// Library/POUs/Trigger/MC_SetTriggerError/Structures/SetTriggerErrorRecvData
{attribute 'pack_mode' := '1'} 
// ------------------------------------------------------------------------- 
//  SRCI Robot Library                                                
// ------------------------------------------------------------------------- 
//                                                                           
//  Object:      SetTriggerErrorRecvData                                       
//  Author:      Thorsten Brach                                                
//  Date:        2024-08-03
//
//  Description:                                              
//   
//                                                                           
//  Copyright: 
//    (C) 2024 Thorsten Brach. All rights reserved                                                                                                                                            
//             Licensed under the LGPL-3.0 license.
//                                                                           
//  Disclaimer:                                                                           
//    This project is provided without any guarantee and can be used for   
//    private and commercial purposes. Any use is at the user’s 
//    own risk and responsibility.
//
// -------------------------------------------------------------------------
TYPE SetTriggerErrorRecvData EXTENDS RspHeader :
STRUCT
  /// Relates to ListenerID >0
  /// Number of successful trigger-based command invocations - For more information refer TO chapter 5.5.12.4
  InvocationCounter : USINT;  
  /// Reserve
  Reserve           : SINT;
  /// Unique system-generated ID of the "Action" when the function is triggered.
  /// • >0: The "Action" is started by the trigger funcrion with identical FollowID.
  /// • <0: The "Action" is stopped by the trigger function with identical FollowID.
  /// For more information see chapter 5.5.12.4 EmitterID, ListenerID, FollowID and OriginID
  OriginID          : INT;
END_STRUCT
END_TYPE

// Library/POUs/Trigger/MC_SetTriggerError/Structures/SetTriggerErrorSendData
{attribute 'pack_mode' := '1'}
// ------------------------------------------------------------------------- 
//  SRCI Robot Library                                                
// ------------------------------------------------------------------------- 
//                                                                           
//  Object:      SetTriggerErrorSendData                                       
//  Author:      Thorsten Brach                                                
//  Date:        2024-08-03
//
//  Description:                                              
//   
//                                                                           
//  Copyright: 
//    (C) 2024 Thorsten Brach. All rights reserved                                                                                                                                            
//             Licensed under the LGPL-3.0 license.
//                                                                           
//  Disclaimer:                                                                           
//    This project is provided without any guarantee and can be used for   
//    private and commercial purposes. Any use is at the user’s 
//    own risk and responsibility.
//
// -------------------------------------------------------------------------
TYPE SetTriggerErrorSendData EXTENDS CmdHeader: 
STRUCT
  /// ID of Action that will be executed when this command is active
  /// • >0: Start Action - Start executing the Action function with the identical ListenerID.
  /// • <0: Stop Action  -  Stop executing the Action function with the identical ListenerID.
  /// • 0: No trigger (default)-  If no EmitterID is defined, the function will not trigger any Action during its execution
  /// For more information see section Triggers of this chapter or chapter 5.5.12.4.
  EmitterID                  : ARRAY [0..3] OF SINT;  
  /// ID of associated trigger function:
  /// • 0: Immediately (default) - Start executing this function immediately.
  /// • >0: Trigger -  Start executing, when the trigger function with the identical EmitterID is triggered.
  /// Always positive.
  /// For more information, see chapter 5.5.12 Triggers
  ListenerID                 : SINT;
  /// Reserve
  Reserve                    : SINT;
  /// Defines error origin through which the associated Action will be triggered
  Mode                       : SINT;
  /// Defines if parametrization messages are included (relates to Mode 0 to 5)
  /// • FALSE (default): Do not include incorrect parametrization
  /// • TRUE: Include incorrect parametrization
  IncludeParameterValidation : BOOL;
  /// Defines message codes through which the associated Action will be triggered (relates to Mode 6 and 7)
  MessageCodes               : ARRAY [0..RobotLibraryParameter.MESSAGE_CODES_MAX] OF DWORD;  
END_STRUCT
END_TYPE

// Library/POUs/Trigger/MC_SetTriggerLimit/Structures/SetTriggerLimitOutCmd
{attribute 'pack_mode' := '1'} 
// ------------------------------------------------------------------------- 
//  SRCI Robot Library                                                
// ------------------------------------------------------------------------- 
//                                                                           
//  Object:      SetTriggerLimitOutCmd                                       
//  Author:      Thorsten Brach                                                
//  Date:        2024-08-03
//
//  Description:                                              
//   
//                                                                           
//  Copyright: 
//    (C) 2024 Thorsten Brach. All rights reserved                                                                                                                                            
//             Licensed under the LGPL-3.0 license.
//                                                                           
//  Disclaimer:                                                                           
//    This project is provided without any guarantee and can be used for   
//    private and commercial purposes. Any use is at the user’s 
//    own risk and responsibility.
//
// -------------------------------------------------------------------------
TYPE SetTriggerLimitOutCmd :
STRUCT
  /// Unique system-generated ID of the "Action" when the function is triggered.
  /// • >0: The "Action" is started by the trigger function with identical FollowID.
  /// • <0: The "Action" is stopped by the trigger function with identical FollowID.
  /// For more information see chapter 5.5.12.4 EmitterID, ListenerID, FollowID and OriginID
  OriginID               : INT;
  /// Relates to ListenerID >0
  /// Number of successful trigger -based command invocations
  /// For more information refer to chapter 5.5.12.4.
  InvocationCounter      : USINT;
  /// Unique system-generated ID of the trigger function when the function is called by user.
  /// For more information see chapter 5.5.12.4.
  FollowID               : DINT;  
END_STRUCT
END_TYPE

// Library/POUs/Trigger/MC_SetTriggerLimit/Structures/SetTriggerLimitParCmd
{attribute 'pack_mode' := '1'} 
// ------------------------------------------------------------------------- 
//  SRCI Robot Library                                                
// ------------------------------------------------------------------------- 
//                                                                           
//  Object:      SetTriggerLimitParCmd                                       
//  Author:      Thorsten Brach                                                
//  Date:        2024-08-03
//
//  Description:                                              
//   
//                                                                           
//  Copyright: 
//    (C) 2024 Thorsten Brach. All rights reserved                                                                                                                                            
//             Licensed under the LGPL-3.0 license.
//                                                                           
//  Disclaimer:                                                                           
//    This project is provided without any guarantee and can be used for   
//    private and commercial purposes. Any use is at the user’s 
//    own risk and responsibility.
//
// -------------------------------------------------------------------------
TYPE SetTriggerLimitParCmd :
STRUCT
  /// Specifies the trigger event by exceeding of the following limit values (one of the following options must be supported)
  TriggerMode            : TriggerModeLimit;
  /// Determines whether the start condition is evaluated or not.
  /// • FALSE: Start condition is not evaluated (default).
  /// • TRUE: Start condition is evaluated
  EvaluateStartCondition : BOOL;
  /// If the tolerance limits for the respective actual data values from the RC are exceeded, the Action function that will be executed.
  /// For "TriggerMode" 1, 2 and 4 the tolerance limits must be entered as follows:
  /// • [0..5]: relates to axes 1 to 6
  /// • [6..11]: relates to external axes 1 to 6.
  /// For "TriggerMode" 3 the tolerance limits must be entered as follows:
  /// • [0]: Following Error in mm.
  /// • [1..11]: Undefined and not relevant.
  /// For all array entries default: 999999
  Data_1                 : ARRAY[0..11] OF REAL;
  /// If the respective actual data values from the RC are under the defined limit, the Action function will be stopped.
  /// For "TriggerMode" 1, 2 and 4 the tolerance limits must be entered as follows:
  /// • [0..5]: relates to axes 1 to 6.
  /// • [6..11]: relates to external axes 1 to 6.
  /// For "TriggerMode" 3 the tolerance limits must be entered as follows:
  /// • [0]: Following Error in mm.
  /// • [1..11]: Undefined and not relevant.
  /// For all array entries default: 999999
  Data_2                 : ARRAY[0..11] OF REAL;
  /// ID of associated trigger function:
  /// • 0: Immediately (default) - Start executing this function immediately.
  /// • >0: Trigger -  Start executing, when the trigger function with the identical EmitterID is triggered.
  /// Always positive.
  /// For more information, see chapter 5.5.12 Triggers
  ListenerID             : SINT;
  /// ID of the Action function that will be executed when the trigger condition is met
  /// • >0: Start Action        - Start executing the Action function with the identical ListenerID.
  /// • <0: Stop Action         - Stop executing the Action function with the identical ListenerID.
  /// •  0: Undefined (default) - If no EmitterID is defined, the function returns an error message
  /// For more information see chapter 5.5.12.4
  EmitterID              : SINT;   
END_STRUCT
END_TYPE

// Library/POUs/Trigger/MC_SetTriggerLimit/Structures/SetTriggerLimitRecvData
{attribute 'pack_mode' := '1'} 
// ------------------------------------------------------------------------- 
//  SRCI Robot Library                                                
// ------------------------------------------------------------------------- 
//                                                                           
//  Object:      SetTriggerLimitRecvData                                       
//  Author:      Thorsten Brach                                                
//  Date:        2024-08-03
//
//  Description:                                              
//   
//                                                                           
//  Copyright: 
//    (C) 2024 Thorsten Brach. All rights reserved                                                                                                                                            
//             Licensed under the LGPL-3.0 license.
//                                                                           
//  Disclaimer:                                                                           
//    This project is provided without any guarantee and can be used for   
//    private and commercial purposes. Any use is at the user’s 
//    own risk and responsibility.
//
// -------------------------------------------------------------------------
TYPE SetTriggerLimitRecvData EXTENDS RspHeader :
STRUCT
  /// Relates to ListenerID >0
  /// Number of successful trigger -based command invocations
  /// For more information refer to chapter 5.5.12.4.
  InvocationCounter      : USINT;
  /// Reserve
  Reserve                : SINT;
  /// Unique system-generated ID of the "Action" when the function is triggered.
  /// • >0: The "Action" is started by the trigger function with identical FollowID.
  /// • <0: The "Action" is stopped by the trigger function with identical FollowID.
  /// For more information see chapter 5.5.12.4 EmitterID, ListenerID, FollowID and OriginID
  OriginID               : INT;
  /// The respective actual data values from the RC that depend on "TriggerMode".
  Data                   : ARRAY [0..11] OF REAL;  
END_STRUCT
END_TYPE

// Library/POUs/Trigger/MC_SetTriggerLimit/Structures/SetTriggerLimitSendData
{attribute 'pack_mode' := '1'}
// ------------------------------------------------------------------------- 
//  SRCI Robot Library                                                
// ------------------------------------------------------------------------- 
//                                                                           
//  Object:      SetTriggerLimitSendData                                       
//  Author:      Thorsten Brach                                                
//  Date:        2024-08-03
//
//  Description:                                              
//   
//                                                                           
//  Copyright: 
//    (C) 2024 Thorsten Brach. All rights reserved                                                                                                                                            
//             Licensed under the LGPL-3.0 license.
//                                                                           
//  Disclaimer:                                                                           
//    This project is provided without any guarantee and can be used for   
//    private and commercial purposes. Any use is at the user’s 
//    own risk and responsibility.
//
// -------------------------------------------------------------------------
TYPE SetTriggerLimitSendData EXTENDS CmdHeader: 
STRUCT
  /// ID of Action that will be executed when this command is active
  /// • >0: Start Action - Start executing the Action function with the identical ListenerID.
  /// • <0: Stop Action  -  Stop executing the Action function with the identical ListenerID.
  /// • 0: No trigger (default)-  If no EmitterID is defined, the function will not trigger any Action during its execution
  /// For more information see section Triggers of this chapter or chapter 5.5.12.4.
  EmitterID              : ARRAY [0..3] OF SINT;  
  /// ID of associated trigger function:
  /// • 0: Immediately (default) - Start executing this function immediately.
  /// • >0: Trigger -  Start executing, when the trigger function with the identical EmitterID is triggered.
  /// Always positive.
  /// For more information, see chapter 5.5.12 Triggers
  ListenerID             : SINT;
  /// If the tolerance limits for the respective actual data values from the RC are exceeded, the Action function that will be executed.
  /// For "TriggerMode" 1, 2 and 4 the tolerance limits must be entered as follows:
  /// • [0..5]: relates to axes 1 to 6
  /// • [6..11]: relates to external axes 1 to 6.
  /// For "TriggerMode" 3 the tolerance limits must be entered as follows:
  /// • [0]: Following Error in mm.
  /// • [1..11]: Undefined and not relevant.
  /// For all array entries default: 999999
  Data_1                 : ARRAY[0..11] OF REAL;
  /// If the respective actual data values from the RC are under the defined limit, the Action function will be stopped.
  /// For "TriggerMode" 1, 2 and 4 the tolerance limits must be entered as follows:
  /// • [0..5]: relates to axes 1 to 6.
  /// • [6..11]: relates to external axes 1 to 6.
  /// For "TriggerMode" 3 the tolerance limits must be entered as follows:
  /// • [0]: Following Error in mm.
  /// • [1..11]: Undefined and not relevant.
  /// For all array entries default: 999999
  Data_2                 : ARRAY[0..11] OF REAL;
  /// Specifies the trigger event by exceeding of the following limit values (one of the following options must be supported)
  TriggerMode            : SINT;
  /// Determines whether the start condition is evaluated or not.
  /// • FALSE: Start condition is not evaluated (default).
  /// • TRUE: Start condition is evaluated
  EvaluateStartCondition : BOOL;
END_STRUCT
END_TYPE

// Library/POUs/Trigger/MC_SetTriggerMotion/Structures/SetTriggerMotionOutCmd
{attribute 'pack_mode' := '1'} 
// ------------------------------------------------------------------------- 
//  SRCI Robot Library                                                
// ------------------------------------------------------------------------- 
//                                                                           
//  Object:      SetTriggerMotionOutCmd                                       
//  Author:      Thorsten Brach                                                
//  Date:        2024-08-03
//
//  Description:                                              
//   
//                                                                           
//  Copyright: 
//    (C) 2024 Thorsten Brach. All rights reserved                                                                                                                                            
//             Licensed under the LGPL-3.0 license.
//                                                                           
//  Disclaimer:                                                                           
//    This project is provided without any guarantee and can be used for   
//    private and commercial purposes. Any use is at the user’s 
//    own risk and responsibility.
//
// -------------------------------------------------------------------------
TYPE SetTriggerMotionOutCmd :
STRUCT
  /// Unique system-generated ID of the "Action" when the function is triggered.
  /// • >0: The "Action" is started by the trigger function with identical FollowID.
  /// • <0: The "Action" is stopped by the trigger function with identical FollowID.
  /// For more information see chapter 5.5.12.4 EmitterID, ListenerID, FollowID and OriginID
  OriginID               : INT;
  /// Relates to ListenerID >0
  /// Number of successful trigger -based command invocations
  /// For more information refer to chapter 5.5.12.4.
  InvocationCounter      : USINT;
  /// Unique system-generated ID of the trigger function when the function is called by user.
  /// For more information see chapter 5.5.12.4.
  FollowID               : DINT;
END_STRUCT
END_TYPE

// Library/POUs/Trigger/MC_SetTriggerMotion/Structures/SetTriggerMotionParCmd
{attribute 'pack_mode' := '1'} 
// ------------------------------------------------------------------------- 
//  SRCI Robot Library                                                
// ------------------------------------------------------------------------- 
//                                                                           
//  Object:      SetTriggerMotionParCmd                                       
//  Author:      Thorsten Brach                                                
//  Date:        2024-08-03
//
//  Description:                                              
//   
//                                                                           
//  Copyright: 
//    (C) 2024 Thorsten Brach. All rights reserved                                                                                                                                            
//             Licensed under the LGPL-3.0 license.
//                                                                           
//  Disclaimer:                                                                           
//    This project is provided without any guarantee and can be used for   
//    private and commercial purposes. Any use is at the user’s 
//    own risk and responsibility.
//
// -------------------------------------------------------------------------
TYPE SetTriggerMotionParCmd :
STRUCT
  ///Defines the trigger condition on which the related Action function will be started:
  TriggerMode_1          : TriggerCondition;
  /// This parameter depends on the input parameter "TriggerMode_1":
  /// • 1: Distance value of trajectory in %.
  /// • 2: Distance value of trajectory in mm.
  /// • 3: TCP velocity value of reference velocity in %
  /// • 4: TCP velocity value of reference velocity in mm.
  /// • 5: Time in ms
  /// The value of the parameter must be positive  
  TriggerParameter_1     : REAL;
  ///Defines the trigger condition on which the related Action function will be started:
  TriggerMode_2          : TriggerCondition;
  /// This parameter depends on the input parameter "TriggerMode_1":
  /// • 1: Distance value of trajectory in %. 
  /// • 2: Distance value of trajectory in mm.
  /// • 3: TCP velocity value of reference velocity in %
  /// • 4: TCP velocity value of reference velocity in mm.
  /// • 5: Time in ms
  /// The value of the parameter must be positive  
  TriggerParameter_2     : REAL;
  /// ID of associated trigger function:
  /// • 0: Immediately (default) - Start executing this function immediately.
  /// • >0: Trigger -  Start executing, when the trigger function with the identical EmitterID is triggered.
  /// Always positive.
  /// For more information, see chapter 5.5.12 Triggers
  ListenerID             : SINT;
  /// ID of the Action function that will be executed when the trigger condition is met
  /// • >0: Start Action        - Start executing the Action function with the identical ListenerID.
  /// • <0: Stop Action         - Stop executing the Action function with the identical ListenerID.
  /// •  0: Undefined (default) - If no EmitterID is defined, the function returns an error message
  /// For more information see chapter 5.5.12.4
  EmitterID              : SINT;  
END_STRUCT
END_TYPE

// Library/POUs/Trigger/MC_SetTriggerMotion/Structures/SetTriggerMotionRecvData
{attribute 'pack_mode' := '1'} 
// ------------------------------------------------------------------------- 
//  SRCI Robot Library                                                
// ------------------------------------------------------------------------- 
//                                                                           
//  Object:      SetTriggerMotionRecvData                                       
//  Author:      Thorsten Brach                                                
//  Date:        2024-08-03
//
//  Description:                                              
//   
//                                                                           
//  Copyright: 
//    (C) 2024 Thorsten Brach. All rights reserved                                                                                                                                            
//             Licensed under the LGPL-3.0 license.
//                                                                           
//  Disclaimer:                                                                           
//    This project is provided without any guarantee and can be used for   
//    private and commercial purposes. Any use is at the user’s 
//    own risk and responsibility.
//
// -------------------------------------------------------------------------
TYPE SetTriggerMotionRecvData EXTENDS RspHeader :
STRUCT
  /// Relates to ListenerID >0
  /// Number of successful trigger -based command invocations
  /// For more information refer to chapter 5.5.12.4.
  InvocationCounter      : USINT;
  /// Reserve
  Reserve                : SINT;
  /// Unique system-generated ID of the "Action" when the function is triggered.
  /// • >0: The "Action" is started by the trigger function with identical FollowID.
  /// • <0: The "Action" is stopped by the trigger function with identical FollowID.
  /// For more information see chapter 5.5.12.4 EmitterID, ListenerID, FollowID and OriginID
  OriginID               : INT;
END_STRUCT
END_TYPE

// Library/POUs/Trigger/MC_SetTriggerMotion/Structures/SetTriggerMotionSendData
{attribute 'pack_mode' := '1'}
// ------------------------------------------------------------------------- 
//  SRCI Robot Library                                                
// ------------------------------------------------------------------------- 
//                                                                           
//  Object:      SetTriggerMotionSendData                                       
//  Author:      Thorsten Brach                                                
//  Date:        2024-08-03
//
//  Description:                                              
//   
//                                                                           
//  Copyright: 
//    (C) 2024 Thorsten Brach. All rights reserved                                                                                                                                            
//             Licensed under the LGPL-3.0 license.
//                                                                           
//  Disclaimer:                                                                           
//    This project is provided without any guarantee and can be used for   
//    private and commercial purposes. Any use is at the user’s 
//    own risk and responsibility.
//
// -------------------------------------------------------------------------
TYPE SetTriggerMotionSendData EXTENDS CmdHeader: 
STRUCT
  /// ID of Action that will be executed when this command is active
  /// • >0: Start Action - Start executing the Action function with the identical ListenerID.
  /// • <0: Stop Action  -  Stop executing the Action function with the identical ListenerID.
  /// • 0: No trigger (default)-  If no EmitterID is defined, the function will not trigger any Action during its execution
  /// For more information see section Triggers of this chapter or chapter 5.5.12.4.
  EmitterID              : ARRAY [0..3] OF SINT;  
  /// ID of associated trigger function:
  /// • 0: Immediately (default) - Start executing this function immediately.
  /// • >0: Trigger -  Start executing, when the trigger function with the identical EmitterID is triggered.
  /// Always positive.
  /// For more information, see chapter 5.5.12 Triggers
  ListenerID             : SINT;
  /// If the tolerance limits for the respective actual data values from the RC are exceeded, the Action function that will be executed.
  /// For "TriggerMode" 1, 2 and 4 the tolerance limits must be entered as follows:
  /// • [0..5]: relates to axes 1 to 6
  /// • [6..11]: relates to external axes 1 to 6.
  /// For "TriggerMode" 3 the tolerance limits must be entered as follows:
  /// • [0]: Following Error in mm.
  /// • [1..11]: Undefined and not relevant.
  /// For all array entries default: 999999
  ///Defines the trigger condition on which the related Action function will be started:
  TriggerMode_1          : SINT;
  ///Defines the trigger condition on which the related Action function will be started:
  TriggerMode_2          : SINT;
  /// This parameter depends on the input parameter "TriggerMode_1":
  /// • 1: Distance value of trajectory in %.
  /// • 2: Distance value of trajectory in mm.
  /// • 3: TCP velocity value of reference velocity in %
  /// • 4: TCP velocity value of reference velocity in mm.
  /// • 5: Time in ms
  /// The value of the parameter must be positive  
  TriggerParameter_1     : REAL;
  /// This parameter depends on the input parameter "TriggerMode_1":
  /// • 1: Distance value of trajectory in %. 
  /// • 2: Distance value of trajectory in mm.
  /// • 3: TCP velocity value of reference velocity in %
  /// • 4: TCP velocity value of reference velocity in mm.
  /// • 5: Time in ms
  /// The value of the parameter must be positive  
  TriggerParameter_2     : REAL;
END_STRUCT
END_TYPE

// Library/POUs/Trigger/MC_SetTriggerRegister/Structures/SetTriggerRegisterOutCmd
{attribute 'pack_mode' := '1'} 
// ------------------------------------------------------------------------- 
//  SRCI Robot Library                                                
// ------------------------------------------------------------------------- 
//                                                                           
//  Object:      SetTriggerRegisterOutCmd                                       
//  Author:      Thorsten Brach                                                
//  Date:        2024-08-03
//
//  Description:                                              
//   
//                                                                           
//  Copyright: 
//    (C) 2024 Thorsten Brach. All rights reserved                                                                                                                                            
//             Licensed under the LGPL-3.0 license.
//                                                                           
//  Disclaimer:                                                                           
//    This project is provided without any guarantee and can be used for   
//    private and commercial purposes. Any use is at the user’s 
//    own risk and responsibility.
//
// -------------------------------------------------------------------------
TYPE SetTriggerRegisterOutCmd :
STRUCT
  /// Unique system-generated ID of the "Action" when the function is triggered.
  /// • >0: The "Action" is started by the trigger function with identical FollowID.
  /// • <0: The "Action" is stopped by the trigger function with identical FollowID.
  /// For more information see chapter 5.5.12.4 EmitterID, ListenerID, FollowID and OriginID
  OriginID               : INT;
  /// Relates to ListenerID >0
  /// Number of successful trigger -based command invocations
  /// For more information refer to chapter 5.5.12.4.
  InvocationCounter      : USINT;
  /// Unique system-generated ID of the trigger function when the function is called by user.
  /// For more information see chapter 5.5.12.4.
  FollowID               : DINT;  
END_STRUCT
END_TYPE

// Library/POUs/Trigger/MC_SetTriggerRegister/Structures/SetTriggerRegisterParCmd
{attribute 'pack_mode' := '1'} 
// ------------------------------------------------------------------------- 
//  SRCI Robot Library                                                
// ------------------------------------------------------------------------- 
//                                                                           
//  Object:      SetTriggerRegisterParCmd                                       
//  Author:      Thorsten Brach                                                
//  Date:        2024-08-03
//
//  Description:                                              
//   
//                                                                           
//  Copyright: 
//    (C) 2024 Thorsten Brach. All rights reserved                                                                                                                                            
//             Licensed under the LGPL-3.0 license.
//                                                                           
//  Disclaimer:                                                                           
//    This project is provided without any guarantee and can be used for   
//    private and commercial purposes. Any use is at the user’s 
//    own risk and responsibility.
//
// -------------------------------------------------------------------------
TYPE SetTriggerRegisterParCmd :
STRUCT
  /// Specifies the trigger event according to Table 6-574.
  /// For more information about registers on the RC see chapters 6.4.4 and 6.4.5.
  TriggerMode            : TriggerModeIo;
  /// Determines whether the start condition is evaluated or not.
  /// • FALSE: Start condition is not evaluated (default).
  /// • TRUE: Start condition is evaluated. 
  EvaluateStartCondition : BOOL;
  /// Depending on "TriggerMode":
  /// • Digital (refers to "TriggerMode" 10-13, 20-23): Specifies the desired byte address of the input or output signal that shall be read.
  /// • Analog/Integer/Real (refers to "TriggerMode" 30-37, 40-47, 50-57, 60- 67): Specifies the target values that shall be read.
  /// For more information about registers refer to Figure 6-206.
  Index                  : USINT;
  /// Depending on "TriggerMode":
  /// • Digital (refers to TriggerMode 10-13,20-23): Specifies the desired bit address of the input or output signal that shall be read.
  /// • Analog/Integer/Real (refers to TriggerMode 30-37, 40-47, 50-57, 60- 67): Not relevant and deactivated for user input.
  /// For more information about registers refer to Figure 6-206
  BitIndex               : USINT;
  /// Reference integer value, for triggering the Action function with the EmitterID.
  /// • Relates to "TriggerMode" 50-57
  IntValue               : ARRAY[1..2] OF INT;
  /// Reference real value, analog input or output value, for triggering the Action function with the EmitterID.
  /// • Relates to "TriggerMode" 30-37, 40-47,60-67
  RealValue              : ARRAY[1..2] OF REAL;
  /// ID of associated trigger function:
  /// • 0: Immediately (default). - Start executing this function immediately.
  /// • >0: Trigger - Start executing, when the trigger function with the identical EmitterID is triggered.
  /// Always positive.
  /// For more information, see chapter 5.5.12 Triggers
  ListenerID             : SINT;
  /// ID of the Action function that will be executed when the trigger condition is met
  /// • >0: Start Action        - Start executing the Action function with the identical ListenerID.
  /// • <0: Stop Action         - Stop executing the Action function with the identical ListenerID.
  /// •  0: Undefined (default) - If no EmitterID is defined, the function returns an error message
  /// For more information see chapter 5.5.12.4
  EmitterID              : SINT;
END_STRUCT
END_TYPE

// Library/POUs/Trigger/MC_SetTriggerRegister/Structures/SetTriggerRegisterRecvData
{attribute 'pack_mode' := '1'} 
// ------------------------------------------------------------------------- 
//  SRCI Robot Library                                                
// ------------------------------------------------------------------------- 
//                                                                           
//  Object:      SetTriggerRegisterRecvData                                       
//  Author:      Thorsten Brach                                                
//  Date:        2024-08-03
//
//  Description:                                              
//   
//                                                                           
//  Copyright: 
//    (C) 2024 Thorsten Brach. All rights reserved                                                                                                                                            
//             Licensed under the LGPL-3.0 license.
//                                                                           
//  Disclaimer:                                                                           
//    This project is provided without any guarantee and can be used for   
//    private and commercial purposes. Any use is at the user’s 
//    own risk and responsibility.
//
// -------------------------------------------------------------------------
TYPE SetTriggerRegisterRecvData EXTENDS RspHeader :
STRUCT
  /// Relates to ListenerID >0
  /// Number of successful trigger -based command invocations
  /// For more information refer to chapter 5.5.12.4.
  InvocationCounter      : USINT;
  /// Reserve
  Reserve                : SINT;
  /// Unique system-generated ID of the "Action" when the function is triggered.
  /// • >0: The "Action" is started by the trigger function with identical FollowID.
  /// • <0: The "Action" is stopped by the trigger function with identical FollowID.
  /// For more information see chapter 5.5.12.4 EmitterID, ListenerID, FollowID and OriginID
  OriginID               : INT;
END_STRUCT
END_TYPE

// Library/POUs/Trigger/MC_SetTriggerRegister/Structures/SetTriggerRegisterSendData
{attribute 'pack_mode' := '1'}
// ------------------------------------------------------------------------- 
//  SRCI Robot Library                                                
// ------------------------------------------------------------------------- 
//                                                                           
//  Object:      SetTriggerRegisterSendData                                       
//  Author:      Thorsten Brach                                                
//  Date:        2024-08-03
//
//  Description:                                              
//   
//                                                                           
//  Copyright: 
//    (C) 2024 Thorsten Brach. All rights reserved                                                                                                                                            
//             Licensed under the LGPL-3.0 license.
//                                                                           
//  Disclaimer:                                                                           
//    This project is provided without any guarantee and can be used for   
//    private and commercial purposes. Any use is at the user’s 
//    own risk and responsibility.
//
// -------------------------------------------------------------------------
TYPE SetTriggerRegisterSendData EXTENDS CmdHeader: 
STRUCT
  /// ID of Action that will be executed when this command is active
  /// • >0: Start Action - Start executing the Action function with the identical ListenerID.
  /// • <0: Stop Action  -  Stop executing the Action function with the identical ListenerID.
  /// • 0: No trigger (default)-  If no EmitterID is defined, the function will not trigger any Action during its execution
  /// For more information see section Triggers of this chapter or chapter 5.5.12.4.
  EmitterID              : ARRAY [0..3] OF SINT;  
  /// ID of associated trigger function:
  /// • 0: Immediately (default) - Start executing this function immediately.
  /// • >0: Trigger -  Start executing, when the trigger function with the identical EmitterID is triggered.
  /// Always positive.
  /// For more information, see chapter 5.5.12 Triggers
  ListenerID             : SINT;
  /// Reserve
  Reserve                : SINT;
  /// Reference integer value, for triggering the Action function with the EmitterID.
  /// • Relates to "TriggerMode" 50-57
  IntValue               : ARRAY[1..2] OF INT;
  /// Reference real value, analog input or output value, for triggering the Action function with the EmitterID.
  /// • Relates to "TriggerMode" 30-37, 40-47,60-67
  RealValue              : ARRAY[1..2] OF REAL;
  /// Specifies the trigger event according to Table 6-574.
  /// For more information about registers on the RC see chapters 6.4.4 and 6.4.5.
  TriggerMode            : SINT;
  /// Depending on "TriggerMode":
  /// • Digital (refers to "TriggerMode" 10-13, 20-23): Specifies the desired byte address of the input or output signal that shall be read.
  /// • Analog/Integer/Real (refers to "TriggerMode" 30-37, 40-47, 50-57, 60- 67): Specifies the target values that shall be read.
  /// For more information about registers refer to Figure 6-206.
  Index                  : USINT;
  /// Depending on "TriggerMode":
  /// • Digital (refers to TriggerMode 10-13,20-23): Specifies the desired bit address of the input or output signal that shall be read.
  /// • Analog/Integer/Real (refers to TriggerMode 30-37, 40-47, 50-57, 60- 67): Not relevant and deactivated for user input.
  /// For more information about registers refer to Figure 6-206
  BitIndex               : USINT;
END_STRUCT
END_TYPE

// Library/POUs/Trigger/MC_SetTriggerUser/Structures/SetTriggerUserOutCmd
{attribute 'pack_mode' := '1'} 
// ------------------------------------------------------------------------- 
//  SRCI Robot Library                                                
// ------------------------------------------------------------------------- 
//                                                                           
//  Object:      SetTriggerUserOutCmd                                       
//  Author:      Thorsten Brach                                                
//  Date:        2024-08-03
//
//  Description:                                              
//   
//                                                                           
//  Copyright: 
//    (C) 2024 Thorsten Brach. All rights reserved                                                                                                                                            
//             Licensed under the LGPL-3.0 license.
//                                                                           
//  Disclaimer:                                                                           
//    This project is provided without any guarantee and can be used for   
//    private and commercial purposes. Any use is at the user’s 
//    own risk and responsibility.
//
// -------------------------------------------------------------------------
TYPE SetTriggerUserOutCmd :
STRUCT
  /// Unique system-generated ID of the "Action" when the function is triggered.
  /// • >0: The "Action" is started by the trigger function with identical FollowID.
  /// • <0: The "Action" is stopped by the trigger function with identical FollowID.
  /// For more information see chapter 5.5.12.4 EmitterID, ListenerID, FollowID and OriginID
  OriginID               : INT;
  /// Relates to ListenerID >0
  /// Number of successful trigger -based command invocations
  /// For more information refer to chapter 5.5.12.4.
  InvocationCounter      : USINT;
  /// Unique system-generated ID of the trigger function when the function is called by user.
  /// For more information see chapter 5.5.12.4.
  FollowID               : DINT;
  
END_STRUCT
END_TYPE

// Library/POUs/Trigger/MC_SetTriggerUser/Structures/SetTriggerUserParCmd
{attribute 'pack_mode' := '1'} 
// ------------------------------------------------------------------------- 
//  SRCI Robot Library                                                
// ------------------------------------------------------------------------- 
//                                                                           
//  Object:      SetTriggerUserParCmd                                       
//  Author:      Thorsten Brach                                                
//  Date:        2024-08-03
//
//  Description:                                              
//   
//                                                                           
//  Copyright: 
//    (C) 2024 Thorsten Brach. All rights reserved                                                                                                                                            
//             Licensed under the LGPL-3.0 license.
//                                                                           
//  Disclaimer:                                                                           
//    This project is provided without any guarantee and can be used for   
//    private and commercial purposes. Any use is at the user’s 
//    own risk and responsibility.
//
// -------------------------------------------------------------------------
TYPE SetTriggerUserParCmd :
STRUCT
  /// ID of the Action function that will be executed when the trigger condition is met
  /// • >0: Start Action        - Start executing the Action function with the identical ListenerID.
  /// • <0: Stop Action         - Stop executing the Action function with the identical ListenerID.
  /// •  0: Undefined (default) - If no EmitterID is defined, the function returns an error message
  /// For more information see chapter 5.5.12.4
  EmitterID              : SINT;
END_STRUCT
END_TYPE

// Library/POUs/Trigger/MC_SetTriggerUser/Structures/SetTriggerUserRecvData
{attribute 'pack_mode' := '1'} 
// ------------------------------------------------------------------------- 
//  SRCI Robot Library                                                
// ------------------------------------------------------------------------- 
//                                                                           
//  Object:      SetTriggerUserRecvData                                       
//  Author:      Thorsten Brach                                                
//  Date:        2024-08-03
//
//  Description:                                              
//   
//                                                                           
//  Copyright: 
//    (C) 2024 Thorsten Brach. All rights reserved                                                                                                                                            
//             Licensed under the LGPL-3.0 license.
//                                                                           
//  Disclaimer:                                                                           
//    This project is provided without any guarantee and can be used for   
//    private and commercial purposes. Any use is at the user’s 
//    own risk and responsibility.
//
// -------------------------------------------------------------------------
TYPE SetTriggerUserRecvData EXTENDS RspHeader :
STRUCT
  /// Relates to ListenerID >0
  /// Number of successful trigger -based command invocations
  /// For more information refer to chapter 5.5.12.4.
  InvocationCounter      : USINT;
  /// Reserve
  Reserve                : SINT;
  /// Unique system-generated ID of the "Action" when the function is triggered.
  /// • >0: The "Action" is started by the trigger function with identical FollowID.
  /// • <0: The "Action" is stopped by the trigger function with identical FollowID.
  /// For more information see chapter 5.5.12.4 EmitterID, ListenerID, FollowID and OriginID
  OriginID               : INT;
END_STRUCT
END_TYPE

// Library/POUs/Trigger/MC_SetTriggerUser/Structures/SetTriggerUserSendData
{attribute 'pack_mode' := '1'}
// ------------------------------------------------------------------------- 
//  SRCI Robot Library                                                
// ------------------------------------------------------------------------- 
//                                                                           
//  Object:      SetTriggerUserSendData                                       
//  Author:      Thorsten Brach                                                
//  Date:        2024-08-03
//
//  Description:                                              
//   
//                                                                           
//  Copyright: 
//    (C) 2024 Thorsten Brach. All rights reserved                                                                                                                                            
//             Licensed under the LGPL-3.0 license.
//                                                                           
//  Disclaimer:                                                                           
//    This project is provided without any guarantee and can be used for   
//    private and commercial purposes. Any use is at the user’s 
//    own risk and responsibility.
//
// -------------------------------------------------------------------------
TYPE SetTriggerUserSendData EXTENDS CmdHeader: 
STRUCT
  /// ID of Action that will be executed when this command is active
  /// • >0: Start Action - Start executing the Action function with the identical ListenerID.
  /// • <0: Stop Action  -  Stop executing the Action function with the identical ListenerID.
  /// • 0: No trigger (default)-  If no EmitterID is defined, the function will not trigger any Action during its execution
  /// For more information see section Triggers of this chapter or chapter 5.5.12.4.
  EmitterID              : ARRAY [0..3] OF SINT;  
  /// ID of associated trigger function:
  /// • 0: Immediately (default) - Start executing this function immediately.
  /// • >0: Trigger -  Start executing, when the trigger function with the identical EmitterID is triggered.
  /// Always positive.
  /// For more information, see chapter 5.5.12 Triggers
  ListenerID             : SINT;
  /// Reserve
  Reserve                : SINT;
  /// Reference integer value, for triggering the Action function with the EmitterID.
  /// • Relates to "TriggerMode" 50-57
  IntValue               : ARRAY[1..2] OF INT;
  /// Reference real value, analog input or output value, for triggering the Action function with the EmitterID.
  /// • Relates to "TriggerMode" 30-37, 40-47,60-67
  RealValue              : ARRAY[1..2] OF REAL;
  /// Specifies the trigger event according to Table 6-574.
  /// For more information about registers on the RC see chapters 6.4.4 and 6.4.5.
  TriggerMode            : SINT;
  /// Depending on "TriggerMode":
  /// • Digital (refers to "TriggerMode" 10-13, 20-23): Specifies the desired byte address of the input or output signal that shall be read.
  /// • Analog/Integer/Real (refers to "TriggerMode" 30-37, 40-47, 50-57, 60- 67): Specifies the target values that shall be read.
  /// For more information about registers refer to Figure 6-206.
  Index                  : USINT;
  /// Depending on "TriggerMode":
  /// • Digital (refers to TriggerMode 10-13,20-23): Specifies the desired bit address of the input or output signal that shall be read.
  /// • Analog/Integer/Real (refers to TriggerMode 30-37, 40-47, 50-57, 60- 67): Not relevant and deactivated for user input.
  /// For more information about registers refer to Figure 6-206
  BitIndex               : USINT;
END_STRUCT
END_TYPE

// Library/POUs/Trigger/MC_WaitForTrigger/Structures/WaitForTriggerOutCmd
{attribute 'pack_mode' := '1'} 
// ------------------------------------------------------------------------- 
//  SRCI Robot Library                                                
// ------------------------------------------------------------------------- 
//                                                                           
//  Object:      WaitForTriggerOutCmd                                       
//  Author:      Thorsten Brach                                                
//  Date:        2024-08-03
//
//  Description:                                              
//   
//                                                                           
//  Copyright: 
//    (C) 2024 Thorsten Brach. All rights reserved                                                                                                                                            
//             Licensed under the LGPL-3.0 license.
//                                                                           
//  Disclaimer:                                                                           
//    This project is provided without any guarantee and can be used for   
//    private and commercial purposes. Any use is at the user’s 
//    own risk and responsibility.
//
// -------------------------------------------------------------------------
TYPE WaitForTriggerOutCmd :
STRUCT
  /// Unique system-generated ID of the "Action" when the function is triggered.
  /// • >0: The "Action" is started by the trigger function with identical FollowID.
  /// • <0: The "Action" is stopped by the trigger function with identical FollowID.
  /// For more information see chapter 5.5.12.4 EmitterID, ListenerID, FollowID and OriginID
  OriginID               : INT;
  /// Relates to ListenerID >0
  /// Number of successful trigger -based command invocations
  /// For more information refer to chapter 5.5.12.4.
  InvocationCounter      : USINT;
END_STRUCT
END_TYPE

// Library/POUs/Trigger/MC_WaitForTrigger/Structures/WaitForTriggerParCmd
{attribute 'pack_mode' := '1'} 
// ------------------------------------------------------------------------- 
//  SRCI Robot Library                                                
// ------------------------------------------------------------------------- 
//                                                                           
//  Object:      WaitForTriggerParCmd                                       
//  Author:      Thorsten Brach                                                
//  Date:        2024-08-03
//
//  Description:                                              
//   
//                                                                           
//  Copyright: 
//    (C) 2024 Thorsten Brach. All rights reserved                                                                                                                                            
//             Licensed under the LGPL-3.0 license.
//                                                                           
//  Disclaimer:                                                                           
//    This project is provided without any guarantee and can be used for   
//    private and commercial purposes. Any use is at the user’s 
//    own risk and responsibility.
//
// -------------------------------------------------------------------------
TYPE WaitForTriggerParCmd :
STRUCT
  /// ID of the Action function that will be executed when the trigger condition is met
  /// • >0: Start Action        - Start executing the Action function with the identical ListenerID.
  /// • <0: Stop Action         - Stop executing the Action function with the identical ListenerID.
  /// •  0: Undefined (default) - If no EmitterID is defined, the function returns an error message
  /// For more information see chapter 5.5.12.4
  EmitterID              : SINT;
  /// ID of associated trigger function:
  /// • 0: Immediately (default) - Start executing this function immediately.
  /// • >0: Trigger -  Start executing, when the trigger function with the identical EmitterID is triggered.
  /// Always positive.
  /// For more information, see chapter 5.5.12 Triggers
  ListenerID             : SINT;
  ///  Defines the time at which the trigger can be reacted to
  /// • 0: Conditional - Trigger signal accepted as soon as the function is BUFFERED
  /// • 1: Absolute - Trigger signal accepted as soon as the function is ACTIVE
  ConditionalWait        : BOOL;
END_STRUCT
END_TYPE

// Library/POUs/Trigger/MC_WaitForTrigger/Structures/WaitForTriggerRecvData
{attribute 'pack_mode' := '1'} 
// ------------------------------------------------------------------------- 
//  SRCI Robot Library                                                
// ------------------------------------------------------------------------- 
//                                                                           
//  Object:      WaitForTriggerRecvData                                       
//  Author:      Thorsten Brach                                                
//  Date:        2024-08-03
//
//  Description:                                              
//   
//                                                                           
//  Copyright: 
//    (C) 2024 Thorsten Brach. All rights reserved                                                                                                                                            
//             Licensed under the LGPL-3.0 license.
//                                                                           
//  Disclaimer:                                                                           
//    This project is provided without any guarantee and can be used for   
//    private and commercial purposes. Any use is at the user’s 
//    own risk and responsibility.
//
// -------------------------------------------------------------------------
TYPE WaitForTriggerRecvData EXTENDS RspHeader :
STRUCT
  /// Relates to ListenerID >0
  /// Number of successful trigger -based command invocations
  /// For more information refer to chapter 5.5.12.4.
  InvocationCounter      : USINT;
  /// Reserve
  Reserve                : SINT;
  /// Unique system-generated ID of the "Action" when the function is triggered.
  /// • >0: The "Action" is started by the trigger function with identical FollowID.
  /// • <0: The "Action" is stopped by the trigger function with identical FollowID.
  /// For more information see chapter 5.5.12.4 EmitterID, ListenerID, FollowID and OriginID
  OriginID               : INT;
END_STRUCT
END_TYPE

// Library/POUs/Trigger/MC_WaitForTrigger/Structures/WaitForTriggerSendData
{attribute 'pack_mode' := '1'}
// ------------------------------------------------------------------------- 
//  SRCI Robot Library                                                
// ------------------------------------------------------------------------- 
//                                                                           
//  Object:      WaitForTriggerSendData                                       
//  Author:      Thorsten Brach                                                
//  Date:        2024-08-03
//
//  Description:                                              
//   
//                                                                           
//  Copyright: 
//    (C) 2024 Thorsten Brach. All rights reserved                                                                                                                                            
//             Licensed under the LGPL-3.0 license.
//                                                                           
//  Disclaimer:                                                                           
//    This project is provided without any guarantee and can be used for   
//    private and commercial purposes. Any use is at the user’s 
//    own risk and responsibility.
//
// -------------------------------------------------------------------------
TYPE WaitForTriggerSendData EXTENDS CmdHeader: 
STRUCT
  /// ID of Action that will be executed when this command is active
  /// • >0: Start Action - Start executing the Action function with the identical ListenerID.
  /// • <0: Stop Action  -  Stop executing the Action function with the identical ListenerID.
  /// • 0: No trigger (default)-  If no EmitterID is defined, the function will not trigger any Action during its execution
  /// For more information see section Triggers of this chapter or chapter 5.5.12.4.
  EmitterID              : ARRAY [0..3] OF SINT;  
  /// ID of associated trigger function:
  /// • 0: Immediately (default) - Start executing this function immediately.
  /// • >0: Trigger -  Start executing, when the trigger function with the identical EmitterID is triggered.
  /// Always positive.
  /// For more information, see chapter 5.5.12 Triggers
  ListenerID             : SINT;
  /// Reserve
  Reserve                : SINT;
  ///  Defines the time at which the trigger can be reacted to
  /// • 0: Conditional - Trigger signal accepted as soon as the function is BUFFERED
  /// • 1: Absolute - Trigger signal accepted as soon as the function is ACTIVE
  ConditionalWait        : BOOL;
END_STRUCT
END_TYPE

// Library/POUs/Trigger/MC_WaitTime/Structures/WaitTimeOutCmd
{attribute 'pack_mode' := '1'} 
// ------------------------------------------------------------------------- 
//  SRCI Robot Library                                                
// ------------------------------------------------------------------------- 
//                                                                           
//  Object:      WaitTimeOutCmd                                       
//  Author:      Thorsten Brach                                                
//  Date:        2024-06-30
//
//  Description:                                              
//   
//                                                                           
//  Copyright: 
//    (C) 2024 Thorsten Brach. All rights reserved                                                                                                                                            
//             Licensed under the LGPL-3.0 license.
//                                                                           
//  Disclaimer:                                                                           
//    This project is provided without any guarantee and can be used for   
//    private and commercial purposes. Any use is at the user’s 
//    own risk and responsibility.
//
// -------------------------------------------------------------------------
TYPE WaitTimeOutCmd :
STRUCT
  /// Current value of time [ms] that has elapsed since processing of the command has started.
  ElapsedTime        : UDINT;  
END_STRUCT
END_TYPE

// Library/POUs/Trigger/MC_WaitTime/Structures/WaitTimeParCmd
{attribute 'pack_mode' := '1'} 
// ------------------------------------------------------------------------- 
//  SRCI Robot Library                                                
// ------------------------------------------------------------------------- 
//                                                                           
//  Object:      WaitTimeParCmd                                       
//  Author:      Thorsten Brach                                                
//  Date:        2024-06-30
//
//  Description:                                              
//   
//                                                                           
//  Copyright: 
//    (C) 2024 Thorsten Brach. All rights reserved                                                                                                                                            
//             Licensed under the LGPL-3.0 license.
//                                                                           
//  Disclaimer:                                                                           
//    This project is provided without any guarantee and can be used for   
//    private and commercial purposes. Any use is at the user’s 
//    own risk and responsibility.
//
// -------------------------------------------------------------------------
TYPE WaitTimeParCmd :
STRUCT
  /// Duration [ms] of the waiting time. The value of the parameter must be positive
  WaitTime           : UDINT;
END_STRUCT
END_TYPE

// Library/POUs/Trigger/MC_WaitTime/Structures/WaitTimeRecvData
{attribute 'pack_mode' := '1'} 
// ------------------------------------------------------------------------- 
//  SRCI Robot Library                                                
// ------------------------------------------------------------------------- 
//                                                                           
//  Object:      WaitTimeRecvData                                       
//  Author:      Thorsten Brach                                                
//  Date:        2024-06-30
//
//  Description:                                              
//   
//                                                                           
//  Copyright: 
//    (C) 2024 Thorsten Brach. All rights reserved                                                                                                                                            
//             Licensed under the LGPL-3.0 license.
//                                                                           
//  Disclaimer:                                                                           
//    This project is provided without any guarantee and can be used for   
//    private and commercial purposes. Any use is at the user’s 
//    own risk and responsibility.
//
// -------------------------------------------------------------------------
TYPE WaitTimeRecvData EXTENDS RspHeader :
STRUCT
  /// Current value of time [ms] that has elapsed since processing of the command has started.
  ElapsedTime : UDINT;
  /// Reserve
  Reserve1    : BYTE;
  /// Reserve
  Reserve2    : BYTE;
  /// Reserve
  Reserve3    : BYTE;
  /// Reserve
  Reserve4    : BYTE;  
END_STRUCT
END_TYPE

// Library/POUs/Trigger/MC_WaitTime/Structures/WaitTimeSendData
{attribute 'pack_mode' := '1'}
// ------------------------------------------------------------------------- 
//  SRCI Robot Library                                                
// ------------------------------------------------------------------------- 
//                                                                           
//  Object:      WaitTimeSendData                                       
//  Author:      Thorsten Brach                                                
//  Date:        2024-06-30
//
//  Description:                                              
//   
//                                                                           
//  Copyright: 
//    (C) 2024 Thorsten Brach. All rights reserved                                                                                                                                            
//             Licensed under the LGPL-3.0 license.
//                                                                           
//  Disclaimer:                                                                           
//    This project is provided without any guarantee and can be used for   
//    private and commercial purposes. Any use is at the user’s 
//    own risk and responsibility.
//
// -------------------------------------------------------------------------
TYPE WaitTimeSendData EXTENDS CmdHeader: 
STRUCT
  /// Duration [ms] of the waiting time. The value of the parameter must be positive
  WaitTime : UDINT;
  /// Reserve
  Reserve1 : BYTE;
  /// Reserve
  Reserve2 : BYTE;
  /// Reserve
  Reserve3 : BYTE;
  /// Reserve
  Reserve4 : BYTE;
END_STRUCT
END_TYPE

// Library/POUs/WorkAreas/MC_ActivateWorkArea/Structures/ActivateWorkAreaOutCmd
{attribute 'pack_mode' := '1'} 
// ------------------------------------------------------------------------- 
//  SRCI Robot Library                                                
// ------------------------------------------------------------------------- 
//                                                                           
//  Object:      ActivateWorkAreaOutCmd                                       
//  Author:      Thorsten Brach                                                
//  Date:        2024-06-01
//
//  Description:                                              
//   
//                                                                           
//  Copyright: 
//    (C) 2024 Thorsten Brach. All rights reserved                                                                                                                                            
//             Licensed under the LGPL-3.0 license.
//                                                                           
//  Disclaimer:                                                                           
//    This project is provided without any guarantee and can be used for   
//    private and commercial purposes. Any use is at the user’s 
//    own risk and responsibility.
//
// -------------------------------------------------------------------------
TYPE ActivateWorkAreaOutCmd :
STRUCT
END_STRUCT
END_TYPE

// Library/POUs/WorkAreas/MC_ActivateWorkArea/Structures/ActivateWorkAreaParCmd
{attribute 'pack_mode' := '1'} 
// ------------------------------------------------------------------------- 
//  SRCI Robot Library                                                
// ------------------------------------------------------------------------- 
//                                                                           
//  Object:      ActivateWorkAreaParCmd                                       
//  Author:      Thorsten Brach                                                
//  Date:        2024-06-01
//
//  Description:                                              
//   
//                                                                           
//  Copyright: 
//    (C) 2024 Thorsten Brach. All rights reserved                                                                                                                                            
//             Licensed under the LGPL-3.0 license.
//                                                                           
//  Disclaimer:                                                                           
//    This project is provided without any guarantee and can be used for   
//    private and commercial purposes. Any use is at the user’s 
//    own risk and responsibility.
//
// -------------------------------------------------------------------------
TYPE ActivateWorkAreaParCmd :
STRUCT
  /// Index of the robot work area to be activated
  /// • 0 (default)..254
  WorkAreaNo         : USINT;
  /// Set to activate work area defined by Index.
  /// Reset to deactivate work area defined by Index.
  ActivateArea       : BOOL;
END_STRUCT
END_TYPE

// Library/POUs/WorkAreas/MC_ActivateWorkArea/Structures/ActivateWorkAreaRecvData
{attribute 'pack_mode' := '1'} 
// ------------------------------------------------------------------------- 
//  SRCI Robot Library                                                
// ------------------------------------------------------------------------- 
//                                                                           
//  Object:      ActivateWorkAreaRecvData                                       
//  Author:      Thorsten Brach                                                
//  Date:        2024-06-01
//
//  Description:                                              
//   
//                                                                           
//  Copyright: 
//    (C) 2024 Thorsten Brach. All rights reserved                                                                                                                                            
//             Licensed under the LGPL-3.0 license.
//                                                                           
//  Disclaimer:                                                                           
//    This project is provided without any guarantee and can be used for   
//    private and commercial purposes. Any use is at the user’s 
//    own risk and responsibility.
//
// -------------------------------------------------------------------------
TYPE ActivateWorkAreaRecvData EXTENDS RspHeader :
STRUCT
END_STRUCT
END_TYPE

// Library/POUs/WorkAreas/MC_ActivateWorkArea/Structures/ActivateWorkAreaSendData
{attribute 'pack_mode' := '1'}
// ------------------------------------------------------------------------- 
//  SRCI Robot Library                                                
// ------------------------------------------------------------------------- 
//                                                                           
//  Object:      ActivateWorkAreaParCmd                                       
//  Author:      Thorsten Brach                                                
//  Date:        2024-06-01
//
//  Description:                                              
//   
//                                                                           
//  Copyright: 
//    (C) 2024 Thorsten Brach. All rights reserved                                                                                                                                            
//             Licensed under the LGPL-3.0 license.
//                                                                           
//  Disclaimer:                                                                           
//    This project is provided without any guarantee and can be used for   
//    private and commercial purposes. Any use is at the user’s 
//    own risk and responsibility.
//
// -------------------------------------------------------------------------
TYPE ActivateWorkAreaSendData EXTENDS CmdHeader:   
STRUCT  
  /// Index of the robot work area to be activated
  /// • 0 (default)..254
  WorkAreaNo         : USINT;
  /// Set to activate work area defined by Index.
  /// Reset to deactivate work area defined by Index.
  ActivateArea       : BOOL;
END_STRUCT
END_TYPE

// Library/POUs/WorkAreas/MC_MonitorWorkArea/Structures/MonitorWorkAreaOutCmd
{attribute 'pack_mode' := '1'} 
// ------------------------------------------------------------------------- 
//  SRCI Robot Library                                                
// ------------------------------------------------------------------------- 
//                                                                           
//  Object:      MonitorWorkAreaOutCmd                                       
//  Author:      Thorsten Brach                                                
//  Date:        2024-06-22
//
//  Description:                                              
//   
//                                                                           
//  Copyright: 
//    (C) 2024 Thorsten Brach. All rights reserved                                                                                                                                            
//             Licensed under the LGPL-3.0 license.
//                                                                           
//  Disclaimer:                                                                           
//    This project is provided without any guarantee and can be used for   
//    private and commercial purposes. Any use is at the user’s 
//    own risk and responsibility.
//
// -------------------------------------------------------------------------
TYPE MonitorWorkAreaOutCmd :
STRUCT
  /// Bits return TRUE when work area defined by Index is active
  ActivationState    : WORD;
  /// Bits return TRUE when violation is reported.
  MonitoringState    : WORD;  
END_STRUCT
END_TYPE

// Library/POUs/WorkAreas/MC_MonitorWorkArea/Structures/MonitorWorkAreaParCmd
{attribute 'pack_mode' := '1'} 
// ------------------------------------------------------------------------- 
//  SRCI Robot Library                                                
// ------------------------------------------------------------------------- 
//                                                                           
//  Object:      MonitorWorkAreaParCmd                                       
//  Author:      Thorsten Brach                                                
//  Date:        2024-06-22
//
//  Description:                                              
//   
//                                                                           
//  Copyright: 
//    (C) 2024 Thorsten Brach. All rights reserved                                                                                                                                            
//             Licensed under the LGPL-3.0 license.
//                                                                           
//  Disclaimer:                                                                           
//    This project is provided without any guarantee and can be used for   
//    private and commercial purposes. Any use is at the user’s 
//    own risk and responsibility.
//
// -------------------------------------------------------------------------
TYPE MonitorWorkAreaParCmd :
STRUCT
  /// Index of robot work area to be monitored
  /// • 0 (default)..254
  WorkAreaNo         : USINT;
END_STRUCT
END_TYPE

// Library/POUs/WorkAreas/MC_MonitorWorkArea/Structures/MonitorWorkAreaRecvData
{attribute 'pack_mode' := '1'} 
// ------------------------------------------------------------------------- 
//  SRCI Robot Library                                                
// ------------------------------------------------------------------------- 
//                                                                           
//  Object:      MonitorWorkAreaRecvData                                       
//  Author:      Thorsten Brach                                                
//  Date:        2024-06-22
//
//  Description:                                              
//   
//                                                                           
//  Copyright: 
//    (C) 2024 Thorsten Brach. All rights reserved                                                                                                                                            
//             Licensed under the LGPL-3.0 license.
//                                                                           
//  Disclaimer:                                                                           
//    This project is provided without any guarantee and can be used for   
//    private and commercial purposes. Any use is at the user’s 
//    own risk and responsibility.
//
// -------------------------------------------------------------------------
TYPE MonitorWorkAreaRecvData EXTENDS RspHeader :
STRUCT
  /// Bits return TRUE when work area defined by Index is active
  ActivationState    : WORD;
  /// Bits return TRUE when violation is reported.
  MonitoringState    : WORD;    
END_STRUCT
END_TYPE

// Library/POUs/WorkAreas/MC_MonitorWorkArea/Structures/MonitorWorkAreaSendData
{attribute 'pack_mode' := '1'}
// ------------------------------------------------------------------------- 
//  SRCI Robot Library                                                
// ------------------------------------------------------------------------- 
//                                                                           
//  Object:      MonitorWorkAreaSendData                                       
//  Author:      Thorsten Brach                                                
//  Date:        2024-06-22
//
//  Description:                                              
//   
//                                                                           
//  Copyright: 
//    (C) 2024 Thorsten Brach. All rights reserved                                                                                                                                            
//             Licensed under the LGPL-3.0 license.
//                                                                           
//  Disclaimer:                                                                           
//    This project is provided without any guarantee and can be used for   
//    private and commercial purposes. Any use is at the user’s 
//    own risk and responsibility.
//
// -------------------------------------------------------------------------
TYPE MonitorWorkAreaSendData EXTENDS CmdHeader: 
STRUCT
  /// Set TRUE to activate monitoring of work areas
  Enable             : BOOL;
  /// Index of robot work area to be monitored
  /// • 0 (default)..254
  WorkAreaNo         : USINT;
END_STRUCT
END_TYPE

// Library/POUs/WorkAreas/MC_ReadWorkArea/Structures/ReadWorkAreaOutCmd
{attribute 'pack_mode' := '1'} 
// ------------------------------------------------------------------------- 
//  SRCI Robot Library                                                
// ------------------------------------------------------------------------- 
//                                                                           
//  Object:      ReadWorkAreaOutCmd                                       
//  Author:      Thorsten Brach                                                
//  Date:        2024-08-09
//
//  Description:                                              
//   
//                                                                           
//  Copyright: 
//    (C) 2024 Thorsten Brach. All rights reserved                                                                                                                                            
//             Licensed under the LGPL-3.0 license.
//                                                                           
//  Disclaimer:                                                                           
//    This project is provided without any guarantee and can be used for   
//    private and commercial purposes. Any use is at the user’s 
//    own risk and responsibility.
//
// -------------------------------------------------------------------------
TYPE ReadWorkAreaOutCmd :
STRUCT
  /// Index of the robot work area
  WorkAreaNoReturn       : USINT;
  /// Data specific to the work area requested by Index.
  WorkAreaData           : RobotWorkArea;
END_STRUCT
END_TYPE

// Library/POUs/WorkAreas/MC_ReadWorkArea/Structures/ReadWorkAreaParCmd
{attribute 'pack_mode' := '1'} 
// ------------------------------------------------------------------------- 
//  SRCI Robot Library                                                
// ------------------------------------------------------------------------- 
//                                                                           
//  Object:      ReadWorkAreaParCmd                                       
//  Author:      Thorsten Brach                                                
//  Date:        2024-08-09
//
//  Description:                                              
//   
//                                                                           
//  Copyright: 
//    (C) 2024 Thorsten Brach. All rights reserved                                                                                                                                            
//             Licensed under the LGPL-3.0 license.
//                                                                           
//  Disclaimer:                                                                           
//    This project is provided without any guarantee and can be used for   
//    private and commercial purposes. Any use is at the user’s 
//    own risk and responsibility.
//
// -------------------------------------------------------------------------
TYPE ReadWorkAreaParCmd :
STRUCT
  /// Index of the robot work area
  /// • 0 (default)..254
  WorkAreaNo             : USINT;
END_STRUCT
END_TYPE

// Library/POUs/WorkAreas/MC_ReadWorkArea/Structures/ReadWorkAreaRecvData
{attribute 'pack_mode' := '1'} 
// ------------------------------------------------------------------------- 
//  SRCI Robot Library                                                
// ------------------------------------------------------------------------- 
//                                                                           
//  Object:      ReadWorkAreaRecvData                                       
//  Author:      Thorsten Brach                                                
//  Date:        2024-08-09
//
//  Description:                                              
//   
//                                                                           
//  Copyright: 
//    (C) 2024 Thorsten Brach. All rights reserved                                                                                                                                            
//             Licensed under the LGPL-3.0 license.
//                                                                           
//  Disclaimer:                                                                           
//    This project is provided without any guarantee and can be used for   
//    private and commercial purposes. Any use is at the user’s 
//    own risk and responsibility.
//
// -------------------------------------------------------------------------
TYPE ReadWorkAreaRecvData EXTENDS RspHeader :
STRUCT
  /// Reserve
  Reserve          : BYTE;
  /// Index of the robot work area
  WorkAreaNoReturn : USINT;
  /// Data specific to the work area requested by Index.
  WorkAreaData     : RobotWorkArea;
  /// ToDo
  DataChanged      : BOOL;
END_STRUCT
END_TYPE

// Library/POUs/WorkAreas/MC_ReadWorkArea/Structures/ReadWorkAreaSendData
{attribute 'pack_mode' := '1'}
// ------------------------------------------------------------------------- 
//  SRCI Robot Library                                                
// ------------------------------------------------------------------------- 
//                                                                           
//  Object:      ReadWorkAreaSendData                                       
//  Author:      Thorsten Brach                                                
//  Date:        2024-08-09
//
//  Description:                                              
//   
//                                                                           
//  Copyright: 
//    (C) 2024 Thorsten Brach. All rights reserved                                                                                                                                            
//             Licensed under the LGPL-3.0 license.
//                                                                           
//  Disclaimer:                                                                           
//    This project is provided without any guarantee and can be used for   
//    private and commercial purposes. Any use is at the user’s 
//    own risk and responsibility.
//
// -------------------------------------------------------------------------
TYPE ReadWorkAreaSendData EXTENDS CmdHeader: 
STRUCT
  /// Index of the robot work area
  /// • 0 (default)..254
  WorkAreaNo             : USINT;
END_STRUCT
END_TYPE

// Library/POUs/WorkAreas/MC_WriteWorkArea/Structures/WriteWorkAreaOutCmd
{attribute 'pack_mode' := '1'} 
// ------------------------------------------------------------------------- 
//  SRCI Robot Library                                                
// ------------------------------------------------------------------------- 
//                                                                           
//  Object:      WriteWorkAreaOutCmd                                       
//  Author:      Thorsten Brach                                                
//  Date:        2024-08-08
//
//  Description:                                              
//   
//                                                                           
//  Copyright: 
//    (C) 2024 Thorsten Brach. All rights reserved                                                                                                                                            
//             Licensed under the LGPL-3.0 license.
//                                                                           
//  Disclaimer:                                                                           
//    This project is provided without any guarantee and can be used for   
//    private and commercial purposes. Any use is at the user’s 
//    own risk and responsibility.
//
// -------------------------------------------------------------------------
TYPE WriteWorkAreaOutCmd :
STRUCT
END_STRUCT
END_TYPE

// Library/POUs/WorkAreas/MC_WriteWorkArea/Structures/WriteWorkAreaParCmd
{attribute 'pack_mode' := '1'} 
// ------------------------------------------------------------------------- 
//  SRCI Robot Library                                                
// ------------------------------------------------------------------------- 
//                                                                           
//  Object:      WriteWorkAreaParCmd                                       
//  Author:      Thorsten Brach                                                
//  Date:        2024-08-08
//
//  Description:                                              
//   
//                                                                           
//  Copyright: 
//    (C) 2024 Thorsten Brach. All rights reserved                                                                                                                                            
//             Licensed under the LGPL-3.0 license.
//                                                                           
//  Disclaimer:                                                                           
//    This project is provided without any guarantee and can be used for   
//    private and commercial purposes. Any use is at the user’s 
//    own risk and responsibility.
//
// -------------------------------------------------------------------------
TYPE WriteWorkAreaParCmd :
STRUCT
  /// Index of the robot work area
  /// • 0 (default)..254
  WorkAreaNo         : USINT;
  /// Data specific to the work area requested by Index.
  WorkAreaData       : RobotWorkArea;
END_STRUCT
END_TYPE

// Library/POUs/WorkAreas/MC_WriteWorkArea/Structures/WriteWorkAreaRecvData
{attribute 'pack_mode' := '1'} 
// ------------------------------------------------------------------------- 
//  SRCI Robot Library                                                
// ------------------------------------------------------------------------- 
//                                                                           
//  Object:      WriteWorkAreaRecvData                                       
//  Author:      Thorsten Brach                                                
//  Date:        2024-08-08
//
//  Description:                                              
//   
//                                                                           
//  Copyright: 
//    (C) 2024 Thorsten Brach. All rights reserved                                                                                                                                            
//             Licensed under the LGPL-3.0 license.
//                                                                           
//  Disclaimer:                                                                           
//    This project is provided without any guarantee and can be used for   
//    private and commercial purposes. Any use is at the user’s 
//    own risk and responsibility.
//
// -------------------------------------------------------------------------
TYPE WriteWorkAreaRecvData EXTENDS RspHeader :
STRUCT
END_STRUCT
END_TYPE

// Library/POUs/WorkAreas/MC_WriteWorkArea/Structures/WriteWorkAreaSendData
{attribute 'pack_mode' := '1'}
// ------------------------------------------------------------------------- 
//  SRCI Robot Library                                                
// ------------------------------------------------------------------------- 
//                                                                           
//  Object:      WriteWorkAreaSendData                                       
//  Author:      Thorsten Brach                                                
//  Date:        2024-08-08
//
//  Description:                                              
//   
//                                                                           
//  Copyright: 
//    (C) 2024 Thorsten Brach. All rights reserved                                                                                                                                            
//             Licensed under the LGPL-3.0 license.
//                                                                           
//  Disclaimer:                                                                           
//    This project is provided without any guarantee and can be used for   
//    private and commercial purposes. Any use is at the user’s 
//    own risk and responsibility.
//
// -------------------------------------------------------------------------
TYPE WriteWorkAreaSendData EXTENDS CmdHeader: 
STRUCT
  /// Reserve
  Reserve           : BYTE;
  /// Index of the robot work area
  /// • 0 (default)..254
  WorkAreaNo         : USINT;
  /// Data specific to the work area requested by Index.
  WorkAreaData       : RobotWorkArea;
  /// Data changed 
  DataChanged        : BOOL;
END_STRUCT
END_TYPE

// Library/POUs/Write/MC_WriteAnalogOutput/Structures/WriteAnalogOutputOutCmd
{attribute 'pack_mode' := '1'} 
// ------------------------------------------------------------------------- 
//  SRCI Robot Library                                                
// ------------------------------------------------------------------------- 
//                                                                           
//  Object:      WriteAnalogOutputOutCmd                                       
//  Author:      Thorsten Brach                                                
//  Date:        2024-08-04
//
//  Description:                                              
//   
//                                                                           
//  Copyright: 
//    (C) 2024 Thorsten Brach. All rights reserved                                                                                                                                            
//             Licensed under the LGPL-3.0 license.
//                                                                           
//  Disclaimer:                                                                           
//    This project is provided without any guarantee and can be used for   
//    private and commercial purposes. Any use is at the user’s 
//    own risk and responsibility.
//
// -------------------------------------------------------------------------
TYPE WriteAnalogOutputOutCmd :
STRUCT
  /// Unique system-generated ID of the "Action" when the function is triggered.
  /// • >0: The "Action" is started by the trigger function with identical FollowID.
  /// • <0: The "Action" is stopped by the trigger function with identical FollowID.
  /// For more information see chapter 5.5.12.4.
  OriginID           : INT;
  /// Relates to ListenerID >0 
  /// Number of successful trigger -based command invocations
  /// For more information refer to chapter 5.5.12.4.
  InvocationCounter  : USINT;
END_STRUCT
END_TYPE

// Library/POUs/Write/MC_WriteAnalogOutput/Structures/WriteAnalogOutputParCmd
{attribute 'pack_mode' := '1'} 
// ------------------------------------------------------------------------- 
//  SRCI Robot Library                                                
// ------------------------------------------------------------------------- 
//                                                                           
//  Object:      WriteAnalogOutputParCmd                                       
//  Author:      Thorsten Brach                                                
//  Date:        2024-08-04
//
//  Description:                                              
//   
//                                                                           
//  Copyright: 
//    (C) 2024 Thorsten Brach. All rights reserved                                                                                                                                            
//             Licensed under the LGPL-3.0 license.
//                                                                           
//  Disclaimer:                                                                           
//    This project is provided without any guarantee and can be used for   
//    private and commercial purposes. Any use is at the user’s 
//    own risk and responsibility.
//
// -------------------------------------------------------------------------
TYPE WriteAnalogOutputParCmd :
STRUCT
  /// Number of the analog input 1..32
  Index              : USINT;
  /// Value of analog output
  Value              : REAL;
  /// Unit of set Value:
  Unit               : UnitType;
  /// Set TRUE to prioritize the execution of this command in the defined target sequence.             
  HighPriority       : BOOL;
  /// ID of associated trigger function:
  /// •  0: No Trigger (default)  No trigger related behavior
  /// • >0: Trigger - Start executing when the trigger function with the identical EmitterID is triggered.
  /// Always positive.
  /// For more information, see chapter 5.5.12 Triggers
  ListenerID         : SINT;
END_STRUCT
END_TYPE

// Library/POUs/Write/MC_WriteAnalogOutput/Structures/WriteAnalogOutputRecvData
{attribute 'pack_mode' := '1'} 
// ------------------------------------------------------------------------- 
//  SRCI Robot Library                                                
// ------------------------------------------------------------------------- 
//                                                                           
//  Object:      WriteAnalogOutputRecvData                                       
//  Author:      Thorsten Brach                                                
//  Date:        2024-08-04
//
//  Description:                                              
//   
//                                                                           
//  Copyright: 
//    (C) 2024 Thorsten Brach. All rights reserved                                                                                                                                            
//             Licensed under the LGPL-3.0 license.
//                                                                           
//  Disclaimer:                                                                           
//    This project is provided without any guarantee and can be used for   
//    private and commercial purposes. Any use is at the user’s 
//    own risk and responsibility.
//
// -------------------------------------------------------------------------
TYPE WriteAnalogOutputRecvData EXTENDS RspHeader :
STRUCT
  /// Relates to ListenerID >0
  /// Number of successful trigger-based command invocations - For more information refer TO chapter 5.5.12.4
  InvocationCounter : USINT;  
  /// Reserve
  Reserve           : SINT;
  /// Unique system-generated ID of the "Action" when the function is triggered.
  /// • >0: The "Action" is started by the trigger funcrion with identical FollowID.
  /// • <0: The "Action" is stopped by the trigger function with identical FollowID.
  /// For more information see chapter 5.5.12.4 EmitterID, ListenerID, FollowID and OriginID
  OriginID          : INT;
END_STRUCT
END_TYPE

